# B&R Automation Studio project TD52 (part 115)

### Module_HA.var - HalIO Package variables
```iecst
(********************************************************************
 * COPYRIGHT -- INNIO Company
 ********************************************************************
 * Package: HAL_IO
 * File: HAL_IO.var
 * Author: 105046866
 * Created: August 23, 2011
 ********************************************************************
 * Variables of package HAL_IO
 ********************************************************************)
VAR
	bPlantComm_interrupted : BOOL := FALSE; (*Plant Communication Interrupted*)
	szGM1_DeviceName : STRING[30] := ''; (*Device name from I/O Module gasmixer 1*)
	szGM2_DeviceName : STRING[30] := ''; (*Device name from I/O Module gasmixer 2*)
	VIS2MM : tVIS2MM;
	MM2VIS : tMM2VIS;
END_VAR
VAR CONSTANT
	READY_FOR_NEW_ENTRY : UINT := 65535;
	W_0mA : INT := 00000; (* Value 0mA *)
	W_2mA : INT := 03276; (* Value 2mA *)
	W_3mA : INT := 04914; (* Value 3mA *)
	W_4mA : INT := 06552; (* Value 4mA *)
	W_20mA : INT := 32760; (* Value 20mA *)
	W_2mA_UR20 : INT := 02765; (* Value 2mA *)
	W_3mA_UR20 : INT := 04147; (* Value 3mA *)
	W_4mA_UR20 : INT := 05530; (* Value 4mA *)
	W_20mA_UR20 : INT := 27648; (* Value 20mA *)
	W_20_5mA_UR20 : INT := 28340; (* Value 20.5mA *)
END_VAR
VAR
	Station : ARRAY[0..149] OF StationCfg_typ;
	StationIO : ARRAY[0..149] OF ModulOK_typ;
	xEngType : EngType; (*engine type*)
	pm : Para_HA_struct;
	Para : Para_HA_struct;
	ParaFactoryDefault : Para_HA_struct := (0);
	ModGrpNrError : UINT;
	ModGrpNrMax : UINT;
	ModNrError : UINT;
	ModNrMax : UINT;
	NodeNrError : UINT;
	bAllModulesOK : BOOL; (*all IO modules are OK*)
	bAllCfgDataOK : BOOL; (*all IO config data are OK*)
	CANDevGo : ARRAY[0..1] OF USINT; (* startup parameter for CAN devices *)
	ECANDevGo : USINT;
	CMSmain_Init : CMSmain;
	CMSmain_Init2 : CMSmain;
	CMSinit_Init : CMSinit;
	CANopen_error : UINT;
	CANopen_CMS : CANopen;
	bGnlTrip : BOOL;
	bGnlTrip1 : BOOL;
	bGnlTrip2 : BOOL;
	bGnlTrip3 : BOOL;
	bGnlWarning : BOOL;
	IN_HA : IN_HA_struct;
	OUT_HA : OUT_HA_struct;
	xGT_CH4 : HALioExtern_Type;
	xGT_H2 : HALioExtern_Type;
	xGT_O2 : HALioExtern_Type;
	xVol_GT : HALioExtern_Type;
	xT_GT : HALioExtern_Type;
	xPr_GT_Gas : HALioExtern_Type;
	xGT_CV : HALioExtern_Type;
	xPr_GT_Suct : HALioExtern_Type;
	xP_Red_Norm : HALioExtern_Type;
	xPr_EngLubOil : HALioExtern_Type;
	xPr_ECW : HALioExtern_Type;
	xPr_Ch_P2s : HALioExtern_Type;
	xPr_Ch_P2 : HALioExtern_Type;
	xPr_CC : HALioExtern_Type;
	ucDevSequencer : USINT;
	CMSexit_Init : CMSexit;
	xPr_EOF_DiffMon : HALioExtern_Type;
	xT_HW_Re : HALioExtern_Type;
	xT_HW_ReAfEC : HALioExtern_Type;
	xT_HW_Su : HALioExtern_Type;
	xCA_IgnP_Set : HALioExtern_Type;
	xDPr_AirFilt_A : HALioExtern_Type;
	xDPr_AirFilt_B : HALioExtern_Type;
	xN_TCHP : HALioExtern_Type;
	xN_TCHP_A : HALioExtern_Type;
	xN_TCHP_B : HALioExtern_Type;
	xN_TCLP : HALioExtern_Type;
	xN_TCLP_A : HALioExtern_Type;
	xN_TCLP_B : HALioExtern_Type;
	xDPr_AirFilt : HALioExtern_Type; (*engine air inlet filter difference pressure*)
	xPr_Ch_P1LP_A : HALioExtern_Type; (* charge pressure before  low press TC*)
	xPr_Ch_P1LP_B : HALioExtern_Type; (* charge pressure before  low press TC*)
	xPr_Ch_P1HP : HALioExtern_Type; (* charge pressure before high press TC*)
	xPr_Ch_P1HP_A : HALioExtern_Type; (* charge pressure before high press TC*)
	xPr_Ch_P1HP_B : HALioExtern_Type; (* charge pressure before high press TC*)
	xPr_PC : HALioExtern_Type;
	xPr_PC_Diff : HALioExtern_Type;
	xPr_Baro : HALioExtern_Type;
	xPr_GT1 : HALioExtern_Type;
	xP_Act_AO : HALioExtern_Type;
	xP_Set_ExtAI_Norm : HALioExtern_Type;
	xP_Red_AI_Norm : HALioExtern_Type;
	xCustAnaIn : ARRAY[0..120] OF HALioExtern_Type;
	xN_Set_ExtAI_Norm : HALioExtern_Type;
	xCtr_CustOut : ARRAY[0..45] OF HALioExtern_Type;
	xCustAnaOut : ARRAY[0..60] OF HALioExtern_Type;
	bNoInitDetected : BOOL := FALSE; (*allways true, except 1cycle on init up*)
	xPr_Ch_P2bFA : HALioExtern_Type;
	xPr_Ch_P2HP : HALioExtern_Type;
	xPr_Ch_P2HP_A : HALioExtern_Type;
	xPr_Ch_P2HP_B : HALioExtern_Type;
	xPr_Ch_P2LP : HALioExtern_Type;
	xPr_Ch_P2LP_A : HALioExtern_Type;
	xPr_Ch_P2LP_B : HALioExtern_Type;
	xPr_Ch_P2_A : HALioExtern_Type;
	xPr_Ch_P2_B : HALioExtern_Type;
	xPr_Ch_P2s_A : HALioExtern_Type;
	xPr_Ch_P2s_B : HALioExtern_Type;
	xPr_PCGT : HALioExtern_Type;
	CANDevGo_InBuffer : ARRAY[0..32] OF CanDeviceGo;
	bMMD_SynchDO : ARRAY[0..2] OF BOOL; (* feedback synch DO *)
	bCANbusoff : BOOL;
	bQuitCANbusoff : BOOL;
	bCANbusoff2 : BOOL;
	bQuitCANbusoff2 : BOOL;
	xPr_HW_Su_LT : HALioExtern_Type;
	xPr_HW_Su_HT : HALioExtern_Type;
	xPr_MGT_a_Filt : HALioExtern_Type;
	xPr_PCGT_Out : HALioExtern_Type;
	xPr_GR_I : HALioExtern_Type;
	xPr_GR_II : HALioExtern_Type;
	xPr_PCGT_sp : HALioExtern_Type;
	xPr_MGT_sp : HALioExtern_Type;
	xF_GenBear_DE1 : HALioExtern_Type;
	xF_GenBear_DE2 : HALioExtern_Type;
	xF_GenBear_NDE1 : HALioExtern_Type;
	xF_GenBear_NDE2 : HALioExtern_Type;
	xPr_ECWaEng : HALioExtern_Type;
	xPr_EOF_After : HALioExtern_Type;
	xPr_TC_EOF_Before : HALioExtern_Type;
	xFlow_OilSkid_DE : HALioExtern_Type;
	xFlow_OilSkid_NDE : HALioExtern_Type;
	xLev_OilSkid_Tank : HALioExtern_Type;
	xPr_OilSkid_HP_NDE : HALioExtern_Type;
	xPr_OilSkid_HP_DE : HALioExtern_Type;
	xT_OilSkid_Supply : HALioExtern_Type;
	xT_OilSkid_Tank : HALioExtern_Type;
	xPr_f_BbFilt : HALioExtern_Type;
	xPr_f_BbFilt_A : HALioExtern_Type;
	xPr_f_BbFilt_B : HALioExtern_Type;
	xPr_a_BbFilt : HALioExtern_Type;
	xPr_a_BbFilt_A : HALioExtern_Type;
	xPr_a_BbFilt_B : HALioExtern_Type;
	xPr_AirStarter_Tank : HALioExtern_Type;
	xPr_AirStarter_Supply : HALioExtern_Type;
	szHalIOErrInfo1 : STRING[99];
	szHalIOErrInfo2 : STRING[99];
	szHalIOErrInfo3 : STRING[99];
	xPos_InlLou1 : HALioExtern_Type;
	xPos_InlLou2 : HALioExtern_Type;
	xPos_OutlLou1 : HALioExtern_Type;
	xPos_OutlLou2 : HALioExtern_Type;
	xPos_CircLou1 : HALioExtern_Type;
	xPos_CircLou2 : HALioExtern_Type;
	xPrDiff_ER : HALioExtern_Type;
	xPos_HW_ReValve : HALioExtern_Type;
	xPos_HW_EC_ReValve : HALioExtern_Type;
	xPos_ChC_Valve : HALioExtern_Type;
	xP_Heat : HALioExtern_Type;
	xPr_EO_Mod_Out : HALioExtern_Type;
	xPr_HW_Re_LT : HALioExtern_Type;
	xPr_HW_Re_HT : HALioExtern_Type;
	xPr_HW_Re_PreH_ECW : HALioExtern_Type;
	xPr_HW_Re_PreH_EO : HALioExtern_Type;
	xPr_OFUbFilt : HALioExtern_Type;
	xPr_OFUaFilt : HALioExtern_Type;
	xPr_OFUbCentrifuge : HALioExtern_Type;
	xP_DEIE : HALioExtern_Type;
	szMMUsynch1_Path : STRING[30];
	szMMUsynch2_Path : STRING[30];
	xPr_TCO : HALioExtern_Type;
	xP_Mns_AnaIn : HALioExtern_Type; (*V4.4 Netzbezugsregler 01*)
	xCtr_Mns_Anain_Setp_W_ext : HALioExtern_Type; (*V4.4 Netzbezugsregler 01*)
	xPF_GenC_SetEU : HALioExtern_Type; (* Power factor setpoint (COS PHI) from EU *)
	xQ_GenC_SetEU : HALioExtern_Type; (* Reactive power setpoint from EU *)
	xQLim_GenC_SetEU : HALioExtern_Type; (* Reactive power limit setpoint from EU *)
	xQU_GenC_Set : HALioExtern_Type; (* Voltage setpoint for reactive power control from EU *)
	xP_GenC_SetEU : HALioExtern_Type; (* Power setpoint from EU *)
	xPLim_GenC_SetEU : HALioExtern_Type; (* Power limit setpoint from EU *)
	xU_SetExtAI_Norm : HALioExtern_Type; (* Voltage setpoint *)
	xQ_Droop_Set : HALioExtern_Type; (* Reactive power droop offset setpoint *)
	xT_EGbCat : HALioExtern_Type;
	xT_EGaCat : HALioExtern_Type;
	xPr_OXIcat_In : HALioExtern_Type;
	xPr_OXIcat_Out : HALioExtern_Type;
	xPr_EG_Deflag_Fast : HALioExtern_Type;
	ucLoopCnt : USINT; (* loop variable *)
	iCnt_OpHours_old : DINT; (* operating hours counter *) (*OldName:betrieb_h; Cycle:2;*)
	ucSAFICommErrEventMax : USINT; (* CAN SAFI All Modules Communication Error Event Max *)
	usSAFICommErrMaxAll : UINT; (* CAN SAFI All Modules Communication Error Max All *)
	usSAFICommErrMaxCur : UINT; (* CAN SAFI All Modules Communication Error Max Current *)
	usSAFICommErrAvgMax : UINT; (* CAN SAFI All Modules Communication Error Average Max *)
	usSAFICommErrAvgMaxCnt : UINT; (* CAN SAFI All Modules Communication Error Average Counter Max *)
	usSAFIPhaseCntMax : UINT; (* CAN SAFI All Modules Communication Error Average Max *)
	usSAFICommErrMax : ARRAY[0..12] OF UINT; (* CAN SAFI Module Communication Error Max *)
	usSAFICommErrAvg : ARRAY[0..12] OF UINT; (* CAN SAFI Module Communication Error Average *)
	usSAFICommErrAvgCnt : ARRAY[0..12] OF UINT; (* CAN SAFI Module Communication Error Average Counter *)
	usSAFIPhaseCnt : ARRAY[0..12] OF UINT; (* CAN SAFI Modules Communication Phase Count *)
	ucTecJetCommErrEventMax : USINT; (* CAN TecJet All Module Communication Error Event Max *)
	usTecJetCommErrMax : UINT; (* CAN TecJet Module Communication Error Max *)
	usTecJetCommErrMaxAll : UINT; (* CAN TecJet All Modules Communication Error Event Max All *)
	usTecJetCommErrMaxCur : UINT; (* CAN TecJet All Modules Communication Error Event Max Current *)
	usTecJetCommErrAvgMax : UINT; (* CAN TecJet All Modules Communication Error Average Max *)
	usTecJetCommErrSlowAvg : UINT; (* CAN TecJet All Modules Communication Error Slow Average *)
	ucTecJetCommErrSlowMax : USINT; (* CAN TecJet All Modules Communication Error Slow Max *)
	usTecJetSlowPhaseCnt : UINT; (* CAN TecJet All Modules Slow Phase Count *)
	usTecJetFastPhaseCntMax : UINT; (* CAN TecJet All Modules Fast Phase Count Max *)
	usTecJetPhaseCntMax : UINT; (* CAN TecJet All Modules Phase Count Max  *)
	usTecJetCommErrFastAvg : ARRAY[0..4] OF UINT; (* CAN TecJet Module Communication Error Fast Average *)
	usTecJetCommErrFastMax : ARRAY[0..4] OF UINT; (* CAN TecJet Module Communication  Error Fast Max *)
	usTecJetFastPhaseCnt : ARRAY[0..4] OF UINT; (* CAN TecJet Module Communication Fast Phase Count *)
	usKLS98CommErrAvgMax : UINT; (* CAN KLS98 Module Communication Error Average Max *)
	ucKLS98CommErrEventMax : USINT; (* CAN KLS98 Module Communication Error Event Max *)
	ucKLS98CommErrMaxAll : USINT; (* CAN KLS98 Module Communication Error Max All *)
	ucKLS98CommErrMaxCur : USINT; (* CAN KLS98 Module Communication Error Max Current *)
	usKLS98PhaseCntMax : UINT; (* CAN KLS98 Module Communication Phase Count Max*)
	usKLS98CommErrAvg : ARRAY[0..24] OF UINT; (* CAN KLS98 All Module Communication Error Average *)
	ucKLS98CommErrMax : ARRAY[0..24] OF USINT; (* CAN KLS98 All Module Communication Error Max *)
	usKLS98PhaseCnt : ARRAY[0..24] OF UINT; (* CAN KLS98 All Module Communication Phase Count*)
	ucIC900CommErrMax : USINT; (* CAN IC900 Module Communication Error Max *)
	usIC900PhaseCnt : UINT; (* CAN IC900 Module Communication Phase Count *)
	usIC900CommErrAvg : UINT; (* CAN IC900 Module Communication Error Average *)
	ucMonicCommErrMax : USINT; (* CAN Monic Module Communication Error Max *)
	usMonicPhaseCnt : UINT; (* CAN Monic Module Communication Phase Count *)
	usMonicCommErrAvg : UINT; (* CAN Monic Module Communication Error Average *)
	xCO_SCR_EMLine1 : HALioExtern_Type; (*FuB*)
	xFlow_SCR_UreaDosingOut : HALioExtern_Type; (*FuB*)
	xNO2_SCR_EMLine1 : HALioExtern_Type; (*FuB*)
	xNO2_SCR_EMLine2 : HALioExtern_Type; (*FuB*)
	xNO_SCR_EMLine1 : HALioExtern_Type; (*FuB*)
	xNO_SCR_EMLine2 : HALioExtern_Type; (*FuB*)
	xO2_SCR_EMLine1 : HALioExtern_Type; (*FuB*)
	xPr_SCR_CatIn : HALioExtern_Type; (*FuB*)
	xPr_SCR_CatOut : HALioExtern_Type; (*FuB*)
	xPr_SCR_ComprAirSupply : HALioExtern_Type; (*FuB*)
	xPr_SCR_UreaDosingIn : HALioExtern_Type; (*FuB*)
	xPr_SCR_UreaDosingOut : HALioExtern_Type; (*FuB*)
	xT_SCR_CatIn : HALioExtern_Type; (*FuB*)
	xT_SCR_CatOut : HALioExtern_Type; (*FuB*)
	bWatchdogSIM2AR : BOOL; (*Watchdog for WinMOD simulation*)
	xPos_ChC2_Valve : HALioExtern_Type;
	xT_GT_NG : HALioExtern_Type;
	xPr_GT_NG : HALioExtern_Type;
	xVol_GT_NG : HALioExtern_Type;
	xPr_AirST_Engage : HALioExtern_Type;
	xPr_ECWaP1 : HALioExtern_Type;
	xPr_ECWaP2 : HALioExtern_Type;
	iUR20_ModuleStatus_I2009_SXX : USINT := 0;
	iUR20_ModuleStatus_I2009_S01 : ARRAY[0..149] OF USINT;
	iUR20_ModuleStatus_I2009_S02 : ARRAY[0..149] OF USINT;
	iUR20_ModuleStatus_I2009_S03 : ARRAY[0..149] OF USINT;
	iUR20_ModuleStatus_I2009_S04 : ARRAY[0..149] OF USINT;
	iUR20_ModuleStatus_I2009_S05 : ARRAY[0..149] OF USINT;
	iUR20_ModuleStatus_I2009_S06 : ARRAY[0..149] OF USINT;
	iUR20_ModuleStatus_I2009_S07 : ARRAY[0..149] OF USINT;
	iUR20_ModuleStatus_I2009_S08 : ARRAY[0..149] OF USINT;
	iUR20_ModuleStatus_I2009_S09 : ARRAY[0..149] OF USINT;
	iUR20_ModuleStatus_I2009_S0A : ARRAY[0..149] OF USINT;
	iUR20_ModuleStatus_I2009_S0B : ARRAY[0..149] OF USINT;
	iUR20_ModuleStatus_I2009_S0C : ARRAY[0..149] OF USINT;
	iUR20_ModuleStatus_I2009_S0D : ARRAY[0..149] OF USINT;
	iUR20_ModuleStatus_I2009_S0E : ARRAY[0..149] OF USINT;
	iUR20_ModuleStatus_I2009_S0F : ARRAY[0..149] OF USINT;
	iUR20_ModuleStatus_I2009_S10 : ARRAY[0..149] OF USINT;
	bUR20_AllModlesOK : BOOL := 0;
	xLev_SCR_UreaTank : HALioExtern_Type; (*FuB*)
	xPr_ThR2_Inlet : HALioExtern_Type; (*FuB*)
	xPr_ThR2_Outlet : HALioExtern_Type; (*FuB*)
END_VAR
VAR CONSTANT
	iNum_CtrlBatMon : USINT := 4; (*number of control battery monitoring test sets*)
END_VAR
VAR
	rMul_MMD_U_Bus : ARRAY[0..2] OF REAL := [3(0.0)]; (* multiplier bus bar voltage *)
	rMul_MMD_U_Synch : ARRAY[0..2] OF REAL := [3(0.0)]; (* multiplier snchronization voltage *)
	rMul_MMD_U_Gen : ARRAY[0..2] OF REAL := [3(0.0)]; (* multiplier generator voltage *)
	xT_EGaHE1 : HALioExtern_Type := (0); (*V4.14 MultiSignalTemp*)
	xT_EGaHE2 : HALioExtern_Type := (0); (*V4.14 MultiSignalTemp*)
	xT_EGaTC : HALioExtern_Type := (0); (*V4.14 MultiSignalTemp*)
	xT_PlateHE : HALioExtern_Type := (0); (*V4.14 MultiSignalTemp*)
	xL_FreshOilTank : HALioExtern_Type := (0); (*V4.12 2022-112*)
	xL_WasteOilTank : HALioExtern_Type := (0); (*V4.12 2022-112*)
	xL_DayOilTank : HALioExtern_Type := (0); (*V4.12 2022-112*)
	MaxNumIoChannels : UINT;
	ActNumIoChannels : UINT;
	xHALioSignal : ARRAY[0..1299] OF HALioSignal;
	xHALioSignals : ARRAY[1..8,0..1299] OF HALioSignal;
	xHALioSignalsCount : ARRAY[1..8] OF UINT;
	callHALioSignal : BOOL;
	HwOK : BOOL;
	ParOK : BOOL;
	xCtr_ChC_Set : HALioExtern_Type; (* Controller 9 - Charge temperature *)
	xCtr_HWRe_Set : HALioExtern_Type; (* Controller 10 - Return water temperature *)
	xCtr_EC_Set : HALioExtern_Type; (* Controller 11 - Return water temperature after cooler *)
	xER_FC_Set : HALioExtern_Type; (* Controller 12 - Room temperature *)
	xCtr_HWSu_Set : HALioExtern_Type; (* Controller 14 - Supply water temperature *)
	xCtr_ChCV_Set : HALioExtern_Type; (* Controller 15 - Charge temperature ventilation - fan *)
	xCtr_ECW_Set : HALioExtern_Type; (* Controller 16 - Engine cooling water temperature *)
	xCtr_ChCHP_Set : HALioExtern_Type; (* Controller 17 - Charge cooler temperature - high pressure *)
	xCtr_GC_Set : HALioExtern_Type; (* Controller 21 - Gas compressor *)
	xEOVal_LT_Set : HALioExtern_Type; (* Controller 22 - Oil temperature controller low temperature *)
	xCtr_InlLou_Set : HALioExtern_Type; (* Controller 23 - Inlet louvre - Room temperature *)
	xCtr_OutlLou_RT_Set : HALioExtern_Type; (* Controller 24 - Outlet louvre - Room temperature *)
	xCtr_OutlLou_RDP_Set : HALioExtern_Type; (* Controller 25 - Outlet louvre - Room difference pressure *)
	xCtr_CircLou_Set : HALioExtern_Type; (* Controller 26 - Circulation louvre - Intake air temperature *)
	xCtr_CDSu_Set : HALioExtern_Type; (* Controller 27 - Supply water temperature condenser *)
	xCtr_OutlVE_RT_Set : HALioExtern_Type; (* Controller 30 - Outlet air fan - Room temperature *)
	xCtr_OutlVE_RDP_Set : HALioExtern_Type; (* Controller 31 - Outlet air fan - Room difference pressure *)
	xCtr_ChC2_Valve_Set : HALioExtern_Type; (* Controller 34 - Charge temperature before HP TC (T1) *)
	bMMD_Out68Cfg_cust : ARRAY[0..2] OF BOOL; (*1 = Activate the usage of usMMD_Out68Cfg_cust for MMD | 0 = (standard) use serial MMD Output68Cfg *)
	usMMD_Out68Cfg_cust : ARRAY[0..2] OF UINT; (* custom Output68Cfg for MMD *)
	Para_iMainsCfg : ARRAY [0..2] OF USINT; (* Mains voltage measurement config *)
	Para_iGenEarthCfg : ARRAY [0..2] OF USINT; (* Generator voltage measurement - Earthing config *)
	Para_iBusEarthCfg : ARRAY [0..2] OF USINT; (* Busbar voltage measurement    - Earthing config *)
	Para_iSynch1EarthCfg : ARRAY [0..2] OF USINT; (* Synch(1) voltage measurement  - Earthing config *)
	Para_iSynch2EarthCfg : ARRAY [0..2] OF USINT; (* Synch(2) voltage measurement  - Earthing config *)
END_VAR
```

### Program Logical/HalIO/IO_Custom (IEC, version 4.14.0) - HalIO Custom IO

#### IO_CustomCyclic.st - Initialization code
```iecst
(*******************************************************************************
AGGR: custom IO channels	(cyclic)

This code is confidential AND proprietary to the INNIO Company.
It may NOT be used in any form, or reproduced in any manner, without the express
written permission of the INNIO Company.
Copyright, INNIO Company, 2025

- list addidtional customized IO channels

Customized modifications: -
------------------------

History:
-------
V3.99	05-07-2012	Weitzer, 	generated FOR modular software
V4.00	14-02-2014	Weitzer, 	change version number
V4.01	19-02-2015  Weitzer,	add error information strings from IOchannel task
V4.14	06-02-2025  Perktold, 	add possibility for customized mains settings for MMD1 and MMD2

Instructions FOR use:
--------------------
- list IO channels which are configured in the IOcgf.dat data module

Outstandings:
------------

*******************************************************************************)

PROGRAM _CYCLIC

	(* Error information strings *)

	szHalIOErrInfo1;
	szHalIOErrInfo2;
	szHalIOErrInfo3;

	(************************************************************)
	(************** BELOW HERE - JUST FOR EXPERTS ***************)
	(* if you ask yourself if you are an expert -> YOU ARE NOT! *)
	(************************************************************)

	(*********)
	(* MMD 1 *)
	(*********)

	(*MMD customized mains setting *)
	bMMD_Out68Cfg_cust[1]		:= FALSE;			(*1 = Activate the usage of bMMD_Out68Cfg_cust[1] for MMD 1 | 0 = (standard) use serial MMD 1 Output68Cfg *)
	Para_iMainsCfg[1]			:= LIMIT(0, 0, 2);	(*<--- define value here *)
	Para_iGenEarthCfg[1]		:= LIMIT(0, 0, 3);	(*<--- define value here *)
	Para_iBusEarthCfg[1]		:= LIMIT(0, 0, 3);	(*<--- define value here *)
	Para_iSynch1EarthCfg[1]		:= LIMIT(0, 0, 3);	(*<--- define value here *)
	Para_iSynch2EarthCfg[1]		:= LIMIT(0, 0, 3);	(*<--- define value here *)

	(* set customized configuration for Output68Cfg *)
	usMMD_Out68Cfg_cust[1].0	:= NOT Para.bGen3PhaseCircuit_Act[1];	(* BIT 00 - Generator mains configuration					*)
	usMMD_Out68Cfg_cust[1].1	:= FALSE;								(* BIT 01 - Reserved - DONT USE								*)
	usMMD_Out68Cfg_cust[1].2	:= NOT Para.bBus3PhaseCircuit_Act[1];	(* BIT 02 - Busbar configuration							*)
	usMMD_Out68Cfg_cust[1].3	:= FALSE;								(* BIT 03 - Reserved - DONT USE								*)
	usMMD_Out68Cfg_cust[1].4	:= Para_iMainsCfg[1].0;					(* BIT 04 - Mains voltage measurement config				*)
	usMMD_Out68Cfg_cust[1].5	:= Para_iMainsCfg[1].1;					(* BIT 05 - Mains voltage measurement config				*)
	usMMD_Out68Cfg_cust[1].6	:= FALSE;								(* BIT 06 - Reserved - DONT USE								*)
	usMMD_Out68Cfg_cust[1].7	:= FALSE;								(* BIT 07 - Reserved - DONT USE								*)
	usMMD_Out68Cfg_cust[1].8	:= Para_iGenEarthCfg[1].0;				(* BIT 08 - Generator voltage measurement - Earthing config	*)
	usMMD_Out68Cfg_cust[1].9	:= Para_iGenEarthCfg[1].1;				(* BIT 09 - Generator voltage measurement - Earthing config	*)
	usMMD_Out68Cfg_cust[1].10	:= Para_iBusEarthCfg[1].0;				(* BIT 10 - Busbar voltage measurement    - Earthing config *)
	usMMD_Out68Cfg_cust[1].11	:= Para_iBusEarthCfg[1].1;				(* BIT 11 - Busbar voltage measurement    - Earthing config *)
	usMMD_Out68Cfg_cust[1].12	:= Para_iSynch1EarthCfg[1].0;			(* BIT 12 - Synch(1) voltage measurement  - Earthing config *)
	usMMD_Out68Cfg_cust[1].13	:= Para_iSynch1EarthCfg[1].1;			(* BIT 13 - Synch(1) voltage measurement  - Earthing config	*)
	usMMD_Out68Cfg_cust[1].14	:= Para_iSynch2EarthCfg[1].0;			(* BIT 14 - Synch(2) voltage measurement  - Earthing config	*)
	usMMD_Out68Cfg_cust[1].15	:= Para_iSynch2EarthCfg[1].1;			(* BIT 15 - Synch(2) voltage measurement  - Earthing config	*)

	(*********)
	(* MMD 2 *)
	(*********)

	(* customized mains setting *)
	bMMD_Out68Cfg_cust[2]		:= FALSE;			(*1 = Activate the usage of bMMD_Out68Cfg_cust[2] for MMD 2 | 0 = (standard) use serial MMD 2 Output68Cfg *)
	Para_iMainsCfg[2]			:= LIMIT(0, 0, 2);	(*<--- define value here *)
	Para_iGenEarthCfg[2]		:= LIMIT(0, 0, 3);	(*<--- define value here *)
	Para_iBusEarthCfg[2]		:= LIMIT(0, 0, 3);	(*<--- define value here *)
	Para_iSynch1EarthCfg[2]		:= LIMIT(0, 0, 3);	(*<--- define value here *)
	Para_iSynch2EarthCfg[2]		:= LIMIT(0, 0, 3);	(*<--- define value here *)

	(* set customized configuration for Output68Cfg *)
	usMMD_Out68Cfg_cust[2].0	:= NOT Para.bGen3PhaseCircuit_Act[2];	(* BIT 00 - Generator mains configuration					*)
	usMMD_Out68Cfg_cust[2].1	:= FALSE;								(* BIT 01 - Reserved - DONT USE								*)
	usMMD_Out68Cfg_cust[2].2	:= NOT Para.bBus3PhaseCircuit_Act[2];	(* BIT 02 - Busbar configuration							*)
	usMMD_Out68Cfg_cust[2].3	:= FALSE;								(* BIT 03 - Reserved - DONT USE								*)
	usMMD_Out68Cfg_cust[2].4	:= Para_iMainsCfg[2].0;					(* BIT 04 - Mains voltage measurement config				*)
	usMMD_Out68Cfg_cust[2].5	:= Para_iMainsCfg[2].1;					(* BIT 05 - Mains voltage measurement config				*)
	usMMD_Out68Cfg_cust[2].6	:= FALSE;								(* BIT 06 - Reserved - DONT USE								*)
	usMMD_Out68Cfg_cust[2].7	:= FALSE;								(* BIT 07 - Reserved - DONT USE								*)
	usMMD_Out68Cfg_cust[2].8	:= Para_iGenEarthCfg[2].0;				(* BIT 08 - Generator voltage measurement - Earthing config	*)
	usMMD_Out68Cfg_cust[2].9	:= Para_iGenEarthCfg[2].1;				(* BIT 09 - Generator voltage measurement - Earthing config	*)
	usMMD_Out68Cfg_cust[2].10	:= Para_iBusEarthCfg[2].0;				(* BIT 10 - Busbar voltage measurement    - Earthing config *)
	usMMD_Out68Cfg_cust[2].11	:= Para_iBusEarthCfg[2].1;				(* BIT 11 - Busbar voltage measurement    - Earthing config *)
	usMMD_Out68Cfg_cust[2].12	:= Para_iSynch1EarthCfg[2].0;			(* BIT 12 - Synch(1) voltage measurement  - Earthing config *)
	usMMD_Out68Cfg_cust[2].13	:= Para_iSynch1EarthCfg[2].1;			(* BIT 13 - Synch(1) voltage measurement  - Earthing config	*)
	usMMD_Out68Cfg_cust[2].14	:= Para_iSynch2EarthCfg[2].0;			(* BIT 14 - Synch(2) voltage measurement  - Earthing config	*)
	usMMD_Out68Cfg_cust[2].15	:= Para_iSynch2EarthCfg[2].1;			(* BIT 15 - Synch(2) voltage measurement  - Earthing config	*)

END_PROGRAM
```

#### IO_CustomInit.st - Initialization code
```iecst
(*******************************************************************************
AGGR: custom IO channels	(init)

This code is confidential AND proprietary to the INNIO Company.
It may NOT be used in any form, or reproduced in any manner, without the express
written permission of the INNIO Company.
Copyright, INNIO Company, 2019

- list addidtional customized IO channels

Customized modifications: -
------------------------

History:
-------
V3.99	05-07-2012	Weitzer, generated FOR modular software
V4.00	14-02-2014	Weitzer, change version number

Instructions FOR use:
--------------------
- list IO channels which are configured in the IOcgf.dat data module

Outstandings:
------------

*******************************************************************************)

PROGRAM _INIT

;

END_PROGRAM
```

### Program Logical/HalIO/IOchannel (IEC, version 4.25.0) - HalIO read & write IO channel

#### IOchannelCyclic.st - Implementation code
```iecst
(*******************************************************************************
AGGR: read and write IO channels	(cyclic)

This code is confidential and proprietary to the INNIO Company.
It may not be used in any form, or reproduced in any manner, without the express
written permission of the INNIO Company.
Copyright, INNIO Company, 2025

- read out data module with IO configuration
- call fubs to copy IO data from IN and to OUT structures

Customized modifications: -
------------------------

History:
-------
V3.99	05-07-2012	Weitzer, generated for modular software
V3.99.1	20-11-2013  zengerer new customized controller 21-28
V4.00	14-02-2014	Weitzer, change version number
V4.01	22-07-2014	Weitzer, change version number
V4.01.1 10-10-2014	Weitzer, set HW OK bit TRUE --> write outputs in case of HW problems
V4.03	14-01-2015	Weitzer, new IOs added for J920
V4.03.1	04-03-2015  zengerer outputs scaling on customized controller AO
V4.03.2 18-01-2016	Weitzer, correction of rOQS_Conduct & rOQS_Dielect ScalMin/Max
V4.03.3 03-03-2016	Weitzer, set F to 0 Hz when no voltage and engine speed > 600
V4.04.0 20-06-2016	Weitzer, add CustAnaOut[17..50]
		06-10-2016	Perktold,added xPLim_DEIE
		24-10-2016	Weitzer, set F to 0 Hz when no voltage and engine speed < 500
V4.05.0	05-04-2017  lettenb. faststart
V4.05.0 16-05-2017  Denk	 tPr_PCGT_a_Filt.Ai := tPr_PCGT.Ai; switching
		17-11-2017	Arnold	 added angle diff for fast synchronization
		04-12.2017	Messner	 old CAT: T_EGbCat, T_EGaCat scalling added
							 new OXIcat: xPr_OXIcat_In, xPr_OXIcat_Out, xPr_OXIcat_In_Fast added
V4.05.1 14.02.2018	Weitzer, EOP_BWS2 added
V4.05.2 26.03.2018	Farre, 	 Signals removed (PF_CosPCtr_PF1_Ena, PF_CosPCtr_PF2_Ena, PF_CosPCtr_PF3_Ena, PF_CosPCtr_PF4_Ena, PF_CosPCtr_PF5_Ena)
V4.07.0	12.07.2018	Hohensinner,	Added G2 Signals
		09.08.2018	Schmid	 2nd low temperature charge cooling circuit added
		20.09.2018	Schmid	 unused IOs deleted
		17.12.2018	Schmid	 IOs FOR hydraulic ECW pre-heating FOR type 3+4 added
		08.01.2019	Schmid	 IOs for redundant pump control added
		10.01.2019	Schmid	 IOs for boiler failure and seismic alarm added
		14.01.2019	Schmid	 Pr_EG_Deflag_Fast (deflagration detection) fully replaces Pr_OXIcat_In_Fast
		13.03.2019	Hohensinner, 	Added custom filter time constant for LSL_In signal
V4.07.2	15.05.2019	Schmid	 coding guidelines: changed Para.rTi_Filt_LSL_In (datatype REAL) to Para.tiFilt_LSL_In (datatype TIME)
V4.09.0 27.06.2019	Denk	 Added parameter scaling for IO's: T_GT_NG, Pr_GT_NG, Vol_GT_NG
V4.09.1	16.04.2020	Schmid	 bugfix: spare analog input (CustAnaIn) scaling corrected to allow falling slope
V4.10.0	26.05.2020	Schmid	 new IOs XT4 v4.10
V4.10.1 10.05.2021	Weitzer	 System cyclic time viaolation monitoring added
V4.10.2	06.12.2021 	Zengerer ArEventLogWrite_0.  //Bugfix- disable line for PPC900
V4.11.0	16.08.2021	Weitzer	 add UR20 IO systemV4.10.2	06.12.2021 	Zengerer ArEventLogWrite_0.  //Bugfix- disable line for PPC900
V4.11.0	17.12.2021 	Schmid	 IOs for control battery check added
		02-02-2022	Zengerer add CustAnaOut[51..60]
V4.12.0	18.11.2022 	Zengerer add L_FreshOilTank, L_WasteOilTank, L_DayOilTank
		22.01.2023 	Zuschnig Added scaling via parameter for H2 signal
		25.01.2025	shifted some parts to new tasks in slower cyclics
V4.13.0	05.03.2024	Bacci	 Added hardware bypass digital twin - T3 adaptive cranking time
V4.14.0	26.02.2025	Tinello	 added SafetyPLC
V4.25.0 26.11.2025	Bacci	 Safety Function - Insufficient Ventilation (2024-202): ERV digital feedback added
		17.12.2025	Tinello	 added SafetyPLC Phase II

Instructions for use:
--------------------
- IO channels are configured in the IOcgf.dat data module

Outstandings:
------------

*******************************************************************************)

PROGRAM _CYCLIC

	(* Set F to 0 Hz when engine; calculate angle *)
	FOR ucCount := 1 TO 2 DO
		IF tU_L1N[ucCount].Ai = 0 AND tU_L2N[ucCount].Ai = 0 AND tU_L3N[ucCount].Ai = 0 AND IN_HA.rN_EngAct < 500 THEN
			F_MMD[ucCount] := 0;
		END_IF;
		IF ssSynchAngleDeviation[ucCount] > 1800 THEN 	(* angle deviation synchronization  +180° - -180° *)
			OUT_HA.rAng_MMD_Diff[ucCount] 	:= INT_TO_REAL(ssSynchAngleDeviation[ucCount]-3600)/10;
		ELSE
			OUT_HA.rAng_MMD_Diff[ucCount] 	:= INT_TO_REAL(ssSynchAngleDeviation[ucCount])/10;
		END_IF;
	END_FOR;

	//	HwOK := bAllModulesOK;
	HwOK := TRUE;
	bAllCfgDataOK := ParOK;

	(* actual power output *)
	tP_Act_AO.Ao := tP_Act[1].Ai;

	(* Gas pressure pre chamber gas train after filter, variable switch *)
	tPr_PCGT_a_Filt.Ai 			:= tPr_PCGT.Ai;
	tPr_PCGT_a_Filt.Unfilt 		:= tPr_PCGT.Unfilt;
	tPr_PCGT_a_Filt.GoodQual 	:= tPr_PCGT.GoodQual;
	Pr_PCGT_a_Filt;

	(* AI und DI for Gricode *)
	tHA2CU.tSet_LFSMO_DB_COn		:= tSet_LFSMO_DB_COn;
	tHA2CU.tSet_LFSMO_DB_COf		:= tSet_LFSMO_DB_COf;
	tHA2GR.tF_LFSMO_DB				:= tF_LFSMO_DB;
	tHA2CU.tSet_LFSMU_DB_COn		:= tSet_LFSMU_DB_COn;
	tHA2CU.tSet_LFSMU_DB_COf		:= tSet_LFSMU_DB_COf;
	tHA2GR.tF_LFSMU_DB				:= tF_LFSMU_DB;
	tHA2CU.tSet_LFSMO_Droop_COn		:= tSet_LFSMO_Droop_COn;
	tHA2CU.tSet_LFSMO_Droop_COf		:= tSet_LFSMO_Droop_COf;
	tHA2GR.tF_LFSMO_Droop			:= tF_LFSMO_Droop;
	tHA2CU.tSet_LFSMU_Droop_COn		:= tSet_LFSMU_Droop_COn;
	tHA2CU.tSet_LFSMU_Droop_COf		:= tSet_LFSMU_Droop_COf;
	tHA2GR.tF_LFSMU_Droop			:= tF_LFSMU_Droop;
	tHA2CU.tSet_FSMU_Droop_COn		:= tSet_FSMU_Droop_COn;
	tHA2CU.tSet_FSMU_Droop_COf		:= tSet_FSMU_Droop_COf;
	tHA2GR.tF_FSMU_Droop			:= tF_FSMU_Droop;
	tHA2CU.tSet_FSMO_Droop_COn		:=	tSet_FSMO_Droop_COn;
	tHA2CU.tSet_FSMO_Droop_COf		:= tSet_FSMO_Droop_COf;
	tHA2GR.tF_FSMO_Droop			:= tF_FSMO_Droop;
	tHA2CU.tSet_FSMU_DB_COn			:= tSet_FSMU_DB_COn;
	tHA2CU.tSet_FSMU_DB_COf			:= tSet_FSMU_DB_COf;
	tHA2GR.tF_FSMU_DB				:= tF_FSMU_DB;
	tHA2CU.tSet_FSMO_DB_COn			:= tSet_FSMO_DB_COn;
	tHA2CU.tSet_FSMO_DB_COf			:= tSet_FSMO_DB_COf;
	tHA2GR.tF_FSMO_DB				:= tF_FSMO_DB;
	tHA2CU.tSet_FSM_RMC_Up_COn		:=	tSet_FSM_RMC_Up_COn;
	tHA2CU.tSet_FSM_RMC_Up_COf		:= tSet_FSM_RMC_Up_COf;
	tHA2GR.tP_FSM_RMC_Up			:= tP_FSM_RMC_Up;
	tHA2CU.tSet_FSM_RMC_Down_COn	:=	tSet_FSM_RMC_Down_COn;
	tHA2CU.tSet_FSM_RMC_Down_COf	:= tSet_FSM_RMC_Down_COf;
	tHA2GR.tP_FSM_RMC_Down			:= tP_FSM_RMC_Down;
	tHA2CU.tSet_U_Droop_COn			:= tSet_U_Droop_COn;
	tHA2CU.tSet_U_Droop_COf			:= tSet_U_Droop_COf;
	tHA2GR.tU_Droop					:= tU_Droop;
	tHA2CU.tSet_FSM_Rmp_COn			:=	tSet_FSM_Rmp_COn;
	tHA2CU.tSet_FSM_Rmp_COf			:= tSet_FSM_Rmp_COf;
	tHA2GR.tFSM_Rmp_Up				:= tFSM_Rmp_Up;
	tHA2GR.tFSM_Rmp_Down			:= tFSM_Rmp_Down;
	tHA2CU.tSet_F_Ref_FSM_COn		:= tSet_F_Ref_FSM_COn;
	tHA2CU.tSet_F_Ref_FSM_COf		:= tSet_F_Ref_FSM_COf;
	tHA2GR.tF_Ref_FSM				:= tF_Ref_FSM;
	tHA2GR.tJunctionBox_GnlAlm		:= tJunctionBox_GnlAlm;
	tHA2GR.bCheck_HA2GR				:= TRUE;
	tHA2CU.bCheck_HA2CU				:= TRUE;

	(* Opstate 4.7 DO addons *)
	xOpMode(in:= IN_HA.iSt_OpMode);
	tOpMode_NetP.Do		:=	xOpMode.NetP;
	tOpMode_Island.Do	:=	xOpMode.Island;
	tOpMode_Idle.Do		:=	xOpMode.Idle;

	L_FreshOilTank;			tL_FreshOilTank;	xL_FreshOilTank;	(*V4.12 Spec 2022-112*)
	L_WasteOilTank;			tL_WasteOilTank;	xL_WasteOilTank;	(*V4.12 Spec 2022-112*)
	L_DayOilTank;			tL_DayOilTank;		xL_DayOilTank;		(*V4.12 Spec 2022-112*)

	(* V4.12 Spec 2022-112 END *)

	(*new with V4.14 SafetyPlc *)
	tGT1_GV1_Open	:= tGV1_Open;									(* SAFETY PLC *)
	tGT1_GV2_Open	:= tGV1_Open;									(* SAFETY PLC *)
	tGT2_GV1_Open	:= tGV2_Open;									(* SAFETY PLC *)
	tGT2_GV2_Open	:= tGV2_Open;									(* SAFETY PLC *)
	tGT3_GV1_Open	:= tGV3_Open;									(* SAFETY PLC *)
	tGT3_GV2_Open	:= tGV3_Open;									(* SAFETY PLC *)
	tGT4_GV1_Open	:= tGV4_Open;									(* SAFETY PLC *)
	tGT4_GV2_Open	:= tGV4_Open;									(* SAFETY PLC *)

	(*new with V4.25 SafetyPlc *)
	tDCGA_GV1_Open	:= tDCGA_GV_Open;								(* SAFETY PLC *)
	tDCGA_GV2_Open	:= tDCGA_GV_Open;								(* SAFETY PLC *)

(**************************************************)

	(* adjust Analog input filter time constant with a parameter, using .Unfilt and .Ai *)
	xFILTER_R_LSL_In.In		:=	tLSL_In.Unfilt;
	xFILTER_R_LSL_In.Filter	:=	TIME_TO_UINT(Para.tiFilt_LSL_In);
	xFILTER_R_LSL_In();
	tLSL_In.Ai	 			:= 	xFILTER_R_LSL_In.Out;

	(* Hardware bypass digital twin - T3 adaptive cranking time *)
	xTOF_HwBypassDigitalTwin(IN := NOT tGV1_Open.Do AND NOT tGV2_Open.Do AND tEleStarter_Dem.Do, PT := T#6s);
	OUT_HA.bTOF_HwBypassDigitalTwin := xTOF_HwBypassDigitalTwin.Q;

	(* Error information strings *)

	szHalIOErrInfo1 := ErrInfo1;
	szHalIOErrInfo2 := ErrInfo2;
	szHalIOErrInfo3 := ErrInfo3;

	(* System cyclic time viaolation monitoring *)

	(* measure real time execution of code *)
	iSysTime_Diff	 := OUT_HA.iSystemTime - iSysTime_Old;		(* current value *)
	iSysTime_Old	 := OUT_HA.iSystemTime;

	(* generate 1 second tick: prevention of too many Logger entries *)
	TON_SecondTick(IN := (NOT TON_SecondTick.Q AND iSysTime_Diff < 2000), PT := T#998ms);		(* 998ms + 2 times cycle time = 1 sec.*)

	(* start new Logger entry *)
	IF iSysTime_Diff > 2000 AND iSysTime_Diff > iSysTime_DiffMax THEN

		(* increase cycle time violation counter *)
		MM2VIS.iNum_CyleTimeViolCnt := MM2VIS.iNum_CyleTimeViolCnt + 1;

			(* write logger entry *)
			memset(ADR(AddData),0,SIZEOF(AddData));
			nextAdr:= brsstrcpy(ADR(AddData), ADR('Cycle time violation in TC#1 | Event count: '));
			strLen:= brsitoa(MM2VIS.iNum_CyleTimeViolCnt, nextAdr);
			nextAdr:= strcat(ADR(AddData),ADR(' | Execution time: '));
			strLen:= brsitoa((iSysTime_Diff/1000), nextAdr);
			nextAdr:= strcat(ADR(AddData),ADR('ms'));
			ArEventLogWrite_0.Execute:= TRUE;		//Bugfix- disable line for PPC900
			ArEventLogWrite_0();					//Bugfix- disable line for PPC900
			ArEventLogWrite_0.Execute:= FALSE;		//Bugfix- disable line for PPC900
			ArEventLogWrite_0();					//Bugfix- disable line for PPC900

		(* set bit for other functions *)
		bCycleTimeViolTriggered := TRUE;

		(* save last diff compare value *)
		iSysTime_DiffMax := iSysTime_Diff;

	ELSE

		(* reset max values for next event *)
		IF TON_SecondTick.Q THEN
			iSysTime_DiffMax := MIN(iSysTime_Diff,iSysTime_DiffMax);	(* min value *)
		END_IF;

	END_IF;

(**************************************************)
	(* Ventilation mapping *)
	(* inlet louvers open (TRUE = opened / FALSE = no longer opened) *)
	tERV_INL1_Lou_OP.Di;	tERV_INL1_Lou_OP.GoodQual;
	tERV_INL2_Lou_OP.Di;	tERV_INL2_Lou_OP.GoodQual;
	tERV_INL3_Lou_OP.Di;	tERV_INL3_Lou_OP.GoodQual;
	tERV_INL4_Lou_OP.Di;	tERV_INL4_Lou_OP.GoodQual;
	tERV_INL5_Lou_OP.Di;	tERV_INL5_Lou_OP.GoodQual;
	tERV_INL6_Lou_OP.Di;	tERV_INL6_Lou_OP.GoodQual;

	(* inlet louvers close (TRUE = closed / FALSE = no longer closed) *)
	tERV_INL1_Lou_CL.Di;	tERV_INL1_Lou_CL.GoodQual;
	tERV_INL2_Lou_CL.Di;	tERV_INL2_Lou_CL.GoodQual;
	tERV_INL3_Lou_CL.Di;	tERV_INL3_Lou_CL.GoodQual;
	tERV_INL4_Lou_CL.Di;	tERV_INL4_Lou_CL.GoodQual;
	tERV_INL5_Lou_CL.Di;	tERV_INL5_Lou_CL.GoodQual;
	tERV_INL6_Lou_CL.Di;	tERV_INL6_Lou_CL.GoodQual;

	(* outlet louvers open (TRUE = opened / FALSE = no longer opened) *)
	tERV_OTL1_Lou_OP.Di;	tERV_OTL1_Lou_OP.GoodQual;
	tERV_OTL2_Lou_OP.Di;	tERV_OTL2_Lou_OP.GoodQual;
	tERV_OTL3_Lou_OP.Di;	tERV_OTL3_Lou_OP.GoodQual;
	tERV_OTL4_Lou_OP.Di;	tERV_OTL4_Lou_OP.GoodQual;
	tERV_OTL5_Lou_OP.Di;	tERV_OTL5_Lou_OP.GoodQual;
	tERV_OTL6_Lou_OP.Di;	tERV_OTL6_Lou_OP.GoodQual;

	(* outlet louvers close (TRUE = closed / FALSE = no longer closed) *)
	tERV_OTL1_Lou_CL.Di;	tERV_OTL1_Lou_CL.GoodQual;
	tERV_OTL2_Lou_CL.Di;	tERV_OTL2_Lou_CL.GoodQual;
	tERV_OTL3_Lou_CL.Di;	tERV_OTL3_Lou_CL.GoodQual;
	tERV_OTL4_Lou_CL.Di;	tERV_OTL4_Lou_CL.GoodQual;
	tERV_OTL5_Lou_CL.Di;	tERV_OTL5_Lou_CL.GoodQual;
	tERV_OTL6_Lou_CL.Di;	tERV_OTL6_Lou_CL.GoodQual;

	(* Fans in operation (TRUE = in operation / FALSE = not in operation)*)
	tERV_INL1_Fan_Run.Di;	tERV_INL1_Fan_Run.GoodQual;
	tERV_INL2_Fan_Run.Di;	tERV_INL2_Fan_Run.GoodQual;
	tERV_INL3_Fan_Run.Di;	tERV_INL3_Fan_Run.GoodQual;
	tERV_INL4_Fan_Run.Di;	tERV_INL4_Fan_Run.GoodQual;
	tERV_INL5_Fan_Run.Di;	tERV_INL5_Fan_Run.GoodQual;
	tERV_INL6_Fan_Run.Di;	tERV_INL6_Fan_Run.GoodQual;

IF IN_HA.bSafetyPLC_Active OR OUT_HA.bSimWinMOD_Active THEN
	(* Inlet Louvers *)
	(* First group of inlet louver connected to stage 1 *)
	IF tERV_INL1_Lou_OP.GoodQual THEN
		tInAirER_Lou1Opened.Di := tERV_INL1_Lou_OP.Di;
		tInAirER_Lou1Opened.GoodQual := tERV_INL1_Lou_OP.GoodQual;
	END_IF;
	IF tERV_INL1_Lou_CL.GoodQual THEN
		tInAirER_Lou1Closed.Di := tERV_INL1_Lou_CL.Di;
		tInAirER_Lou1Closed.GoodQual := tERV_INL1_Lou_CL.GoodQual;
	END_IF;

	(* Second group of inlet louver connected to stage 2*)
	IF tERV_INL2_Lou_OP.GoodQual THEN
		tInAirER_Lou2Opened.Di := tERV_INL2_Lou_OP.Di;
		tInAirER_Lou2Opened.GoodQual := tERV_INL2_Lou_OP.GoodQual;
	END_IF;
	IF tERV_INL2_Lou_CL.GoodQual THEN
		tInAirER_Lou2Closed.Di := tERV_INL2_Lou_CL.Di;
		tInAirER_Lou2Closed.GoodQual := tERV_INL2_Lou_CL.GoodQual;
	END_IF;

	(* Third group of inlet louver connected to stage 1*)
	IF tERV_INL3_Lou_OP.GoodQual THEN
		tInAirER_Lou1Opened.Di := tInAirER_Lou1Opened.Di AND tERV_INL3_Lou_OP.Di;
	END_IF;
	IF tERV_INL3_Lou_CL.GoodQual THEN
		tInAirER_Lou1Closed.Di := tInAirER_Lou1Closed.Di AND tERV_INL3_Lou_CL.Di;
	END_IF;

	(* Fourth group of inlet louver connected to stage 2*)
	IF tERV_INL4_Lou_OP.GoodQual THEN
		tInAirER_Lou2Opened.Di := tInAirER_Lou2Opened.Di AND tERV_INL4_Lou_OP.Di;
	END_IF;
	IF tERV_INL4_Lou_CL.GoodQual THEN
		tInAirER_Lou2Closed.Di := tInAirER_Lou2Closed.Di AND tERV_INL4_Lou_CL.Di;
	END_IF;

	(* Firth group of inlet louver connected to stage 1*)
	IF tERV_INL5_Lou_OP.GoodQual THEN
		tInAirER_Lou1Opened.Di := tInAirER_Lou1Opened.Di AND tERV_INL5_Lou_OP.Di;
	END_IF;
	IF tERV_INL5_Lou_CL.GoodQual THEN
		tInAirER_Lou1Closed.Di := tInAirER_Lou1Closed.Di AND tERV_INL5_Lou_CL.Di;
	END_IF;

	(* Sixth group of inlet louver connected to stage 2*)
	IF tERV_INL6_Lou_OP.GoodQual THEN
		tInAirER_Lou2Opened.Di := tInAirER_Lou2Opened.Di AND tERV_INL6_Lou_OP.Di;
	END_IF;
	IF tERV_INL6_Lou_CL.GoodQual THEN
		tInAirER_Lou2Closed.Di := tInAirER_Lou2Closed.Di AND tERV_INL6_Lou_CL.Di;
	END_IF;

	(* Outlet Louvers *)
	(* First group of outlet louver *)
	IF tERV_OTL1_Lou_OP.GoodQual THEN
		tOutAirER_LouOpened.Di := tERV_OTL1_Lou_OP.Di;
		tOutAirER_LouOpened.GoodQual := tERV_OTL1_Lou_OP.GoodQual;
	END_IF;
	IF tERV_OTL1_Lou_CL.GoodQual THEN
		tOutAirER_LouClosed.Di := tERV_OTL1_Lou_CL.Di;
		tOutAirER_LouClosed.GoodQual := tERV_OTL1_Lou_CL.GoodQual;
	END_IF;

	(* Second group of outlet louver *)
	IF tERV_OTL2_Lou_OP.GoodQual THEN
		tOutAirER_LouOpened.Di := tOutAirER_LouOpened.Di AND tERV_OTL2_Lou_OP.Di;
	END_IF;
	IF tERV_OTL2_Lou_CL.GoodQual THEN
		tOutAirER_LouClosed.Di := tOutAirER_LouClosed.Di AND tERV_OTL2_Lou_CL.Di;
	END_IF;

	(* Third group of outlet louver *)
	IF tERV_OTL3_Lou_OP.GoodQual THEN
		tOutAirER_LouOpened.Di := tOutAirER_LouOpened.Di AND tERV_OTL3_Lou_OP.Di;
	END_IF;
	IF tERV_OTL3_Lou_CL.GoodQual THEN
		tOutAirER_LouClosed.Di := tOutAirER_LouClosed.Di AND tERV_OTL3_Lou_CL.Di;
	END_IF;

	(* Fourth group of outlet louver *)
	IF tERV_OTL4_Lou_OP.GoodQual THEN
		tOutAirER_LouOpened.Di := tOutAirER_LouOpened.Di AND tERV_OTL4_Lou_OP.Di;
	END_IF;
	IF tERV_OTL4_Lou_CL.GoodQual THEN
		tOutAirER_LouClosed.Di := tOutAirER_LouClosed.Di AND tERV_OTL4_Lou_CL.Di;
	END_IF;

	(* Fifth group of outlet louver *)
	IF tERV_OTL5_Lou_OP.GoodQual THEN
		tOutAirER_LouOpened.Di := tOutAirER_LouOpened.Di AND tERV_OTL5_Lou_OP.Di;
	END_IF;
	IF tERV_OTL5_Lou_CL.GoodQual THEN
		tOutAirER_LouClosed.Di := tOutAirER_LouClosed.Di AND tERV_OTL5_Lou_CL.Di;
	END_IF;

	(* Sixth group of outlet louver *)
	IF tERV_OTL6_Lou_OP.GoodQual THEN
		tOutAirER_LouOpened.Di := tOutAirER_LouOpened.Di AND tERV_OTL6_Lou_OP.Di;
	END_IF;
	IF tERV_OTL6_Lou_CL.GoodQual THEN
		tOutAirER_LouClosed.Di := tOutAirER_LouClosed.Di AND tERV_OTL6_Lou_CL.Di;
	END_IF;
END_IF;

IF IN_HA.bSafetyPLC_Active THEN
	(* Safety loop from SAFETY PLC *)
	tSafetyLoop_EmStop.Di		:= IN_HA.bSafeOUT_SafetyLoop_EmStop;
	tSafetyLoop_EmStop.GoodQual	:= TRUE;

	tSafetyLoop_Eng.Di			:= IN_HA.bSafeOUT_SafetyLoop_Eng;
	tSafetyLoop_Eng.GoodQual	:= TRUE;
END_IF;

(**************************************************)

END_PROGRAM
```
